// TIA Portal V17 export
// export: Created 2023-04-11T11:40:01.6946169Z, ExportSetting WithDefaults, DisplayName Totally Integrated Automation Portal, DisplayVersion V17 Update 3, DisplayName TIA Portal Openness, DisplayVersion V17 Update 3, DisplayName TIA Portal Version Control Interface, DisplayVersion V17, DisplayName SINAMICS Startdrive Advanced, DisplayVersion V17 Update2, DisplayName SINAMICS Startdrive G130, G150, S120, S150, SINAMICS MV, S210, DisplayVersion V17 Update2, DisplayName SINAMICS Startdrive G110M, G120, G120C, G120D, G120P, G115D, DisplayVersion V17 Update2, DisplayName STEP 7 Professional, DisplayVersion V17 Update 3, DisplayName STEP 7 Safety, DisplayVersion V17, DisplayName WinCC UA Professional, DisplayVersion V17 Update 3
TYPE "t_DT_FML_REF"
// stored: IsFailsafeCompliant false
   STRUCT
      InData : Struct
         FHPP : Array[1..8] of Byte;
         FPC : Array[1..8] of Byte;
         FHPPplus : Array[1..10] of DInt;
      END_STRUCT;
      OutData : Struct
         FHPP : Array[1..8] of Byte;
         FPC : Array[1..8] of Byte;
         FHPPplus : Array[1..10] of DInt;
      END_STRUCT;
      DeviceType : String[16];
      MemberID : Int;
      MemberIDmax : Int;
      Done : Bool;
      Err : Bool;
      PNU : Word;
      ActPNU : Word;
      ReqID : Int;
      RespID : Int;
      FPCC_Modus : Byte;
      FPCS_Modus : Byte;
      FPCC_Packet { S7_SetPoint := 'True'} : "t_DT_FML_PRM_FILE";
      FPCS_Packet { S7_SetPoint := 'True'} : "t_DT_FML_PRM_FILE";
      Subindex : Byte;
      ActSubindex : Byte;
      DatatypeWR : Int;
      DatatypeRD : Int;
      ParamValueWR : DInt;
      ParamValueRD : DInt;
   END_STRUCT;
END_TYPE
